// TwinCAT 3 PLC project DB
// ProgramVersion: 3.1.4026.16
// libraries:
//   Tc2_Standard, * (Beckhoff Automation GmbH)
//   Tc2_System, * (Beckhoff Automation GmbH)
//   Tc2_Utilities, * (Beckhoff Automation GmbH)
//   Tc3_Database, * (Beckhoff Automation GmbH)
// project tree:
//   DUTs/ ST_ReadConvDb.TcDUT, ST_WriteDb.TcDUT, ST_ReadDb.TcDUT
//   / PlcTask.TcTTO
//   POUs/ MAIN.TcPOU, PlcExpert.TcPOU, PlcExpertCmd.TcPOU, SqlExpert.TcPOU
// real-time tasks:
//   TASK PlcTask: cycle T#10ms, priority 20, ADS port 350

CONFIGURATION DB
    RESOURCE PLC ON TwinCAT3
        TASK PlcTask(INTERVAL := T#10ms, PRIORITY := 20);
        PROGRAM MAIN WITH PlcTask : MAIN;
    END_RESOURCE
END_CONFIGURATION

// ---- DUTs/ST_ReadConvDb.TcDUT
TYPE ST_ReadConvDb :
STRUCT
	nId			: DINT;
	sMachine	: STRING(20);
	sWorkpiece	: STRING(20);
	dtTimestart	: DT;
	dtTimestop	: DT;
	sDuration	: STRING(255); // interval data type not supported
END_STRUCT
END_TYPE

// ---- DUTs/ST_WriteDb.TcDUT
TYPE ST_WriteDb :
STRUCT
	sMachine	: STRING(20);
	sWorkpiece	: STRING(20);
	dtTimeStart	: DT;
	dtTimeStop	: DT;
END_STRUCT
END_TYPE

// ---- DUTs/ST_ReadDb.TcDUT
TYPE ST_ReadDb :
STRUCT
	nId			: DINT;
	sMachine	: STRING(20);
	sWorkpiece	: STRING(20);
	dtTimestart	: DT;
	dtTimestop	: DT;
END_STRUCT
END_TYPE

// ---- POUs/MAIN.TcPOU
PROGRAM MAIN
VAR
END_VAR

SqlExpert();

END_PROGRAM

// ---- POUs/SqlExpert.TcPOU
PROGRAM SqlExpert
VAR
	// Get local time from operating system
	fbLocalTime				: FB_LocalSystemTime;	
	
	// Database interaction FB
	fbSqlDatabase			: FB_SQLDatabaseEvt(sNetID:='', tTimeout:=T#10S);
	fbSqlCommand 			: FB_SQLCommandEvt(sNetID := '', tTimeout := T#10S);
    fbSqlResult				: FB_SQLResultEvt(sNetID:='', tTimeout:=T#10S);
	
	// SQL command
	fbCmdWrite				: FB_FormatString;
	sMachine				: STRING(255);
	sWorkpiece				: STRING(255);
	sTimeStart				: STRING(255);
	sTimeStop				: STRING(255);
	sCmdWrite				: STRING(1000);
	sCmdRead				: STRING(1000);
	
	// Read data
	stReadConvDb			: ST_ReadConvDb;
	
	// Program state
	nDbState				: INT;
	
	// Record trigger
	bMcRun					: BOOL;
END_VAR

// Timestamp sync
fbLocalTime(
	sNetID:= , 
	bEnable:= TRUE, 
	dwCycle:= , 
	dwOpt:= , 
	tTimeout:= , 
	bValid=> , 
	systemTime=> , 
	tzID=> );

// Value
sMachine := 'Milling';
sWorkpiece := 'Shaft';
	
// String manipulation
fbCmdWrite(
	sFormat:= 'INSERT INTO productionlog (machine, workpiece, timestart, timestop) 
			  VALUES ($'%s$', $'%s$', $'%s$', $'%s$')', 
	arg1:= F_STRING(sMachine), 
	arg2:= F_STRING(sWorkpiece), 
	arg3:= F_STRING(sTimeStart), 
	arg4:= F_STRING(sTimeStop), 
	arg5:= , 
	arg6:= , 
	arg7:= , 
	arg8:= , 
	arg9:= , 
	arg10:= , 
	bError=> , 
	nErrId=> , 
	sOut=> sCmdWrite);

sCmdRead := 'SELECT id, machine, workpiece, timestart, timestop, to_char(duration, $'HH24:MI:SS$'::text) AS duration
   			FROM productionlog
			ORDER BY id DESC
			LIMIT 1';

// Program sequence
CASE nDbState OF
	0 : // Init
		bMcRun := FALSE;
		
		nDbState := nDbState + 10;
		
	10 : // Connect to database
		IF fbSqlDatabase.Connect(hDBID:= 1) THEN
			IF fbSqlDatabase.bError THEN
				nDbState := 1000;
			ELSE
				nDbState := nDbState + 10;
			END_IF
		END_IF
		
	20 : // Init command instance
		IF fbSqlDatabase.CreateCmd(pSQLCommand:= ADR(fbSqlCommand)) THEN
			IF fbSqlDatabase.bError THEN
				nDbState := 1000;
			ELSE
				nDbState := 100;
			END_IF
		END_IF
		
	100 : // Wait machine run
		IF bMcRun THEN
			nDbState := nDbState + 10;
		END_IF
		
	110 : // Record time start
		sTimeStart := CONCAT(CONCAT(MID(STR:= SYSTEMTIME_TO_STRING(fbLocalTime.systemTime), LEN:= 10, POS:= 1),' '),
			MID(STR:= SYSTEMTIME_TO_STRING(fbLocalTime.systemTime), LEN:= 8, POS:= 12));
		
		nDbState := nDbState + 10;
		
	120 : // Wait machine stop
		IF NOT bMcRun THEN
			nDbState := nDbState + 10;
		END_IF
		
	130 : // Record time stop
		sTimeStop := CONCAT(CONCAT(MID(STR:= SYSTEMTIME_TO_STRING(fbLocalTime.systemTime), LEN:= 10, POS:= 1),' '),
			MID(STR:= SYSTEMTIME_TO_STRING(fbLocalTime.systemTime), LEN:= 8, POS:= 12));
		
		nDbState := nDbState + 10;
		
	140 : // Write database
		IF fbSqlCommand.Execute(pSQLCmd:= ADR(sCmdWrite), cbSQLCmd:= SIZEOF(sCmdWrite)) THEN
			IF fbSqlCommand.bError THEN
				nDbState := 1000;
			ELSE
				nDbState := 200;
			END_IF
		END_IF
		
	200 : // Read database
		IF fbSqlCommand.ExecuteDataReturn(pSQLCmd:= ADR(sCmdRead), cbSQLCmd:= SIZEOF(sCmdRead), pSQLDBResult:= ADR(fbSqlResult)) THEN
			IF fbSqlCommand.bError THEN
				nDbState := 1000;
			ELSE
				nDbState := nDbState + 10;
			END_IF
		END_IF		
	
	210 : // Read result
		IF fbSqlResult.Read(
			nStartIndex:= 0, 
			nRecordCount:= 1, 
			pData:= ADR(stReadConvDb), 
			cbData:= SIZEOF(stReadConvDb), 
			bWithVerifying:= TRUE, 
			bDataRelease:= FALSE)
		THEN
			IF fbSqlResult.bError THEN
				nDbState := 1000;
			ELSE
				nDbState := nDbState + 10;
			END_IF
		END_IF
		
	220 : // Release cache (optional)
		IF fbSqlResult.Release() THEN
			IF fbSqlResult.bError THEN
				nDbState := 1000;
			ELSE
				nDbState := 100;
			END_IF
		END_IF		
		
	1000 : // Error handling
			
END_CASE

END_PROGRAM

// ---- POUs/PlcExpert.TcPOU
PROGRAM PlcExpert
VAR
	// Get local time from operating system
	fbLocalTime		: FB_LocalSystemTime;		
	
	// Database write and read FB
	fbPlcDbWrite    : FB_PLCDBWriteEvt(sNetID := '', tTimeout := T#5S);
	fbPlcDbRead    	: FB_PLCDBReadEvt (sNetID := '', tTimeout := T#5S);
	fbPlcDbReadDur 	: FB_PLCDBReadEvt (sNetID := '', tTimeout := T#5S);
	
	// Write and read data
	stWriteDb		: ST_WriteDb;
	stReadDb		: ST_ReadDb;
	stReadConvDb	: ST_ReadConvDb;
	
	// Database column name
	ColumnWrite     : ARRAY[0..3] OF STRING(50);
	ColumnRead     	: ARRAY[0..4] OF STRING(50);
	ColumnConvRead  : ARRAY[0..5] OF STRING(50);	
	
	// Program state
	nDbState		: INT;
	
	// Record trigger
	bMcRun			: BOOL;
END_VAR

// Timestamp sync
fbLocalTime(
	sNetID:= , 
	bEnable:= TRUE, 
	dwCycle:= , 
	dwOpt:= , 
	tTimeout:= , 
	bValid=> , 
	systemTime=> , 
	tzID=> );

// Value
stWriteDb.sMachine := 'Milling';
stWriteDb.sWorkpiece := 'Shaft';

// Column names
ColumnWrite[0] := 'machine';
ColumnWrite[1] := 'workpiece';
ColumnWrite[2] := 'timestart';
ColumnWrite[3] := 'timestop';

ColumnRead[0] := 'id';
ColumnRead[1] := 'machine';
ColumnRead[2] := 'workpiece';
ColumnRead[3] := 'timestart';
ColumnRead[4] := 'timestop';

ColumnConvRead[0] := 'id';
ColumnConvRead[1] := 'machine';
ColumnConvRead[2] := 'workpiece';
ColumnConvRead[3] := 'timestart';
ColumnConvRead[4] := 'timestop';
ColumnConvRead[5] := 'duration';

// Program sequence
CASE nDbState OF
	0 : // Init
		bMcRun := FALSE;
		
		nDbState := nDbState + 10;
		
	10 : // Wait machine run
		IF bMcRun THEN
			nDbState := nDbState + 10;
		END_IF
		
	20 : // Record time start
		stWriteDb.dtTimeStart := SYSTEMTIME_TO_DT(fbLocalTime.systemTime);
		
		nDbState := nDbState + 10;
		
	30 : // Wait machine stop
		IF NOT bMcRun THEN
			nDbState := nDbState + 10;
		END_IF
		
	40 : // Record time stop
		stWriteDb.dtTimeStop := SYSTEMTIME_TO_DT(fbLocalTime.systemTime);
		
		nDbState := nDbState + 10;
		
	50 : // Write database
		IF fbPlcDbWrite.WriteStruct(
    		hDBID:= 1, 
    		sTableName:= 'productionlog', 
    		pRecord:= ADR(stWriteDb), 
    		cbRecord:= SIZEOF(stWriteDb), 
    		pColumnNames:= ADR(ColumnWrite) , 
    		cbColumnNames:= SIZEOF(ColumnWrite))
		THEN
			IF fbPlcDbWrite.bError THEN
				nDbState := 1000; 
			ELSE
				nDbState := 100;
			END_IF
		END_IF		
		
	100 : // Read database
		IF fbPlcDbRead.ReadStruct(
			hDBID:= 1, 
			sTableName:= 'productionlog', 
			pColumnNames:= ADR(ColumnRead), 
			cbColumnNames:= SIZEOF(ColumnRead), 
			sOrderByColumn:= ColumnRead[0], 
			eOrderType:= E_OrderType.DESC, 
			nStartIndex:= 0, 
			nRecordCount:= 1, 
			pData:= ADR(stReadDB), 
			cbData:= SIZEOF(stReadDB))
		THEN
			IF fbPlcDbRead.bError THEN
				nDbState := 1000; 
			ELSE
				nDbState := nDbState + 10;
			END_IF
		END_IF
		
	110 : // Read database with duration
		IF fbPlcDbRead.ReadStruct(
			hDBID:= 1, 
			sTableName:= 'viewinterval', 
			pColumnNames:= ADR(ColumnConvRead), 
			cbColumnNames:= SIZEOF(ColumnConvRead), 
			sOrderByColumn:= ColumnRead[0], 
			eOrderType:= E_OrderType.DESC, 
			nStartIndex:= 0, 
			nRecordCount:= 1, 
			pData:= ADR(stReadConvDb), 
			cbData:= SIZEOF(stReadConvDb))
		THEN
			IF fbPlcDbRead.bError THEN
				nDbState := 1000; 
			ELSE
				nDbState := 0;
			END_IF
		END_IF
		
	1000 : // Error handling
	
END_CASE

END_PROGRAM

// ---- POUs/PlcExpertCmd.TcPOU
PROGRAM PlcExpertCmd
VAR
	// Get local time from operating system
	fbLocalTime		: FB_LocalSystemTime;	
	
	// Database write and read FB
	fbPlcDbCmd		: FB_PLCDBCmdEvt(sNetID := '', tTimeout := T#5S);
	
	// SQL query string
    sCmdWrite     	: STRING (1000); 
	sCmdRead     	: STRING (1000); 
	
	// Write and read data
    stWriteDb     	: ST_WriteDb;
	stReadConvDb	: ST_ReadConvDb;
	nLimit			: UINT := 1;
    aPara         	: ARRAY[0..3] OF ST_ExpParameter;
	stPara			: ST_ExpParameter;
	nRecord			: UDINT;
	
	// Program state
	nDbState		: INT;
	
	// Record trigger
	bMcRun			: BOOL;
END_VAR

// Timestamp sync
fbLocalTime(
	sNetID:= , 
	bEnable:= TRUE, 
	dwCycle:= , 
	dwOpt:= , 
	tTimeout:= , 
	bValid=> , 
	systemTime=> , 
	tzID=> );
	
// Value
stWriteDb.sMachine := 'Milling';
stWriteDb.sWorkpiece := 'Shaft';

// Parameter configuration
aPara[0].sParaName := 'sMachine';    
aPara[0].eParaType := E_ExpParameterType.STRING_;      
aPara[0].nParaSize := 21;

aPara[1].sParaName := 'sWorkpiece';   
aPara[1].eParaType := E_ExpParameterType.STRING_;      
aPara[1].nParaSize := 21;

aPara[2].sParaName := 'dtTimeStart';  
aPara[2].eParaType := E_ExpParameterType.DateTime;      
aPara[2].nParaSize := 4;

aPara[3].sParaName := 'dtTimeStop';  
aPara[3].eParaType := E_ExpParameterType.DateTime;      
aPara[3].nParaSize := 4;

stPara.sParaName := 'nLimit';  
stPara.eParaType := E_ExpParameterType.Int16;      
stPara.nParaSize := 2;

// SQL command
sCmdWrite := 'INSERT INTO productionlog (machine, workpiece, timestart, timestop) 
	VALUES ({sMachine}, {sWorkpiece}, {dtTimeStart}, {dtTimeStop})';
	
sCmdRead := 'SELECT * FROM viewinterval
	ORDER BY id DESC
	LIMIT {nLimit}';

// Program sequence
CASE nDbState OF
	0 : // Init
		bMcRun := FALSE;
		
		nDbState := nDbState + 10;
		
	10 : // Wait machine run
		IF bMcRun THEN
			nDbState := nDbState + 10;
		END_IF
		
	20 : // Record time start
		stWriteDb.dtTimeStart := SYSTEMTIME_TO_DT(fbLocalTime.systemTime);
		
		nDbState := nDbState + 10;
		
	30 : // Wait machine stop
		IF NOT bMcRun THEN
			nDbState := nDbState + 10;
		END_IF
		
	40 : // Record time stop
		stWriteDb.dtTimeStop := SYSTEMTIME_TO_DT(fbLocalTime.systemTime);
		
		nDbState := nDbState + 10;
		
	50 : // Write database
		IF fbPlcDbCmd.Execute(
			hDBID:= 1, 
			pExpression:= ADR(sCmdWrite), 
			cbExpression:= SIZEOF(sCmdWrite), 
			pData:= ADR(stWriteDb), 
			cbData:= SIZEOF(stWriteDb), 
			pParameter:= ADR(aPara), 
			cbParameter:= SIZEOF(aPara)) 
		THEN
			IF fbPlcDbCmd.bError THEN
				nDbState := 1000; 
			ELSE
				nDbState := 100;
			END_IF
		END_IF
	
	100 : // Read database with duration
		IF fbPlcDbCmd.ExecuteDataReturn(
			hDBID:= 1, 
			pExpression:= ADR(sCmdRead), 
			cbExpression:= SIZEOF(sCmdRead), 
			pData:= ADR(nLimit), 
			cbData:= SIZEOF(nLimit), 
			pParameter:= ADR(stPara), 
			cbParameter:= SIZEOF(stPara),
			nStartIndex:= 0, 
			nRecordCount:= 10, 
			pReturnData:= ADR(stReadConvDb), 
			cbReturnData:= SIZEOF(stReadConvDb), 
			pRecords:= ADR(nRecord))
		THEN
			IF fbPlcDbCmd.bError THEN
				nDbState := 1000; 
			ELSE
				nDbState := 0;
			END_IF
		END_IF
		
	1000 : // Error handling
	
END_CASE

END_PROGRAM
